RoboDK station: Simulation copy.rdk

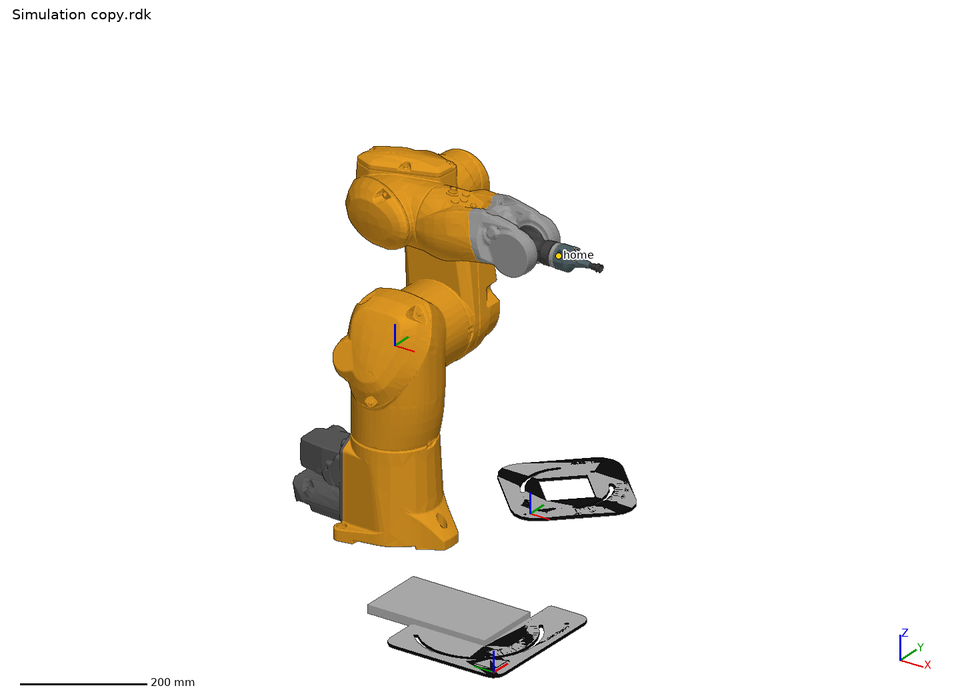
[picture v0: the station drawn from its stored meshes, robots at their saved joint values, targets as dots, program paths as lines]
Station Simulation (saved by RoboDK 5.9.1). Poses are relative to the parent item; angles as X-Y-Z fixed-axis rotations.
  - frame world at (0, 0, 0) mm
    - frame Staubli TX2-40 Base at (0, 0, 0) mm
      - robot Staubli TX2-40: 6 axes, payload 2 kg, reach 515 mm, repeatability 0.02 mm, weight 29 kg
          modified DH rows (alpha deg, a mm, theta deg, d mm): 0, 0, 0, 320; -90, 0, -90, 35; 0, 225, -90, 0; -90, 0, 0, 225; 90, 0, 0, 0; -90, 0, 180, 65
          base shift (0, 0, -320) mm
          joint limits [-180, -180, -180, -270, -180, -270] to [180, 180, 180, 270, 180.5, 270]; home [0, 0, 90, 0, 0, 0]; saved at [0, 0, 90, 0, 0, 0]
        - tool AROB_LWS_VakuumGreifer_14, TCP at (0, 0, 0) mm, size 81.8 x 41.9 x 49.7 mm, geometry from AROB_LWS_VakuumGreifer_14.stp
      - target home (Cartesian target) at (290, 35, 225) mm, rotated rx 0 ry 90 rz 0 deg; joints [0, 0, 90, 0, 0, 0] of Staubli TX2-40
    - frame MagazineFrame at (400, -300, -340) mm, rotated rx 0 ry 0 rz 90 deg
      - object magazinplatte at (100, 100, 0) mm, size 260 x 220 x 5 mm, geometry from AROB_Magazinplatte.stl
      - object jengastuck1 at (72.5, 97.5, 0) mm, rotated rx 0 ry 0 rz 90 deg, size 75 x 25 x 15 mm, geometry from AROB_Jengastuck.stl
      - object jengastuck2 at (97.5, 97.5, 0) mm, rotated rx 0 ry 0 rz 90 deg, size 75 x 25 x 15 mm, geometry from AROB_Jengastuck.stl
      - object jengastuck3 at (122.5, 97.5, 0) mm, rotated rx 0 ry 0 rz 90 deg, size 75 x 25 x 15 mm, geometry from AROB_Jengastuck.stl
      - object jengastuck4 at (147.5, 97.5, 0) mm, rotated rx 0 ry 0 rz 90 deg, size 75 x 25 x 15 mm, geometry from AROB_Jengastuck.stl
      - object jengastuck5 at (172.5, 97.5, 0) mm, rotated rx 0 ry 0 rz 90 deg, size 75 x 25 x 15 mm, geometry from AROB_Jengastuck.stl
      - object jengastuck6 at (72.5, 172.5, 0) mm, rotated rx 0 ry 0 rz 90 deg, size 75 x 25 x 15 mm, geometry from AROB_Jengastuck.stl
      - object jengastuck7 at (97.5, 172.5, 0) mm, rotated rx 0 ry 0 rz 90 deg, size 75 x 25 x 15 mm, geometry from AROB_Jengastuck.stl
      - object jengastuck8 at (122.5, 172.5, 0) mm, rotated rx 0 ry 0 rz 90 deg, size 75 x 25 x 15 mm, geometry from AROB_Jengastuck.stl
      - object jengastuck9 at (147.5, 172.5, 0) mm, rotated rx 0 ry 0 rz 90 deg, size 75 x 25 x 15 mm, geometry from AROB_Jengastuck.stl
      - object jengastuck10 at (172.5, 172.5, 0) mm, rotated rx 0 ry 0 rz 90 deg, size 75 x 25 x 15 mm, geometry from AROB_Jengastuck.stl
      - object jengastuck11 at (72.5, 247.5, 0) mm, rotated rx 0 ry 0 rz 90 deg, size 75 x 25 x 15 mm, geometry from AROB_Jengastuck.stl
      - object jengastuck12 at (97.5, 247.5, 0) mm, rotated rx 0 ry 0 rz 90 deg, size 75 x 25 x 15 mm, geometry from AROB_Jengastuck.stl
      - object jengastuck13 at (122.5, 247.5, 0) mm, rotated rx 0 ry 0 rz 90 deg, size 75 x 25 x 15 mm, geometry from AROB_Jengastuck.stl
      - object jengastuck14 at (147.5, 247.5, 0) mm, rotated rx 0 ry 0 rz 90 deg, size 75 x 25 x 15 mm, geometry from AROB_Jengastuck.stl
      - object jengastuck15 at (172.5, 247.5, 0) mm, rotated rx 0 ry 0 rz 90 deg, size 75 x 25 x 15 mm, geometry from AROB_Jengastuck.stl
    - frame TowerFrame at (120, 200, -340) mm
      - object turmplatte at (0, 100, 0) mm, rotated rx 0 ry 0 rz 45 deg, size 200 x 200 x 5 mm, geometry from AROB_Turmplatte.stl
  - Python program main (listed below)

--- Python program main ---
# main.py

import time
from robodk import robolink

from magazine import Magazine
from tower import Tower
from robot_controller import RobotController
from gripper import Gripper
from jenga_logic import GrabAtPos, ReleaseAtPos

def main():
    # Initialisierung RoboDK API
    rdk = robolink.Robolink()

     # ❗ Kollisionserkennung deaktivieren (nur zum Testen!)
    rdk.setCollisionActive(False)

    # Koordinatenursprünge
    magazine_frame = [330, -100, -300]
    tower_frame = [120, 200, -300]

    # Objekte erzeugen
    magazine = Magazine(magazine_frame)
    tower = Tower(tower_frame)
    robot = RobotController(rdk)
    gripper = Gripper(rdk)

    jenga_pieces = [rdk.Item(f"AROB_Jengastuck{i+1}") for i in range(0,15)]

    for piece in jenga_pieces:
        print(f"Position:{piece.Name()}")



    # Startposition anfahren
    robot.move_to_start()
    robot.move_to_idle()

    # 15 Steine verarbeiten
    for i in range(15):
        source_piece = magazine.get_next_piece()
        source_piece = jenga_pieces[i]
        target_piece = tower.get_next_target(source_piece)

        GrabAtPos(robot, source_piece, gripper)
        ReleaseAtPos(robot, target_piece, gripper)

    # Abschluss
    robot.move_to_start()

if __name__ == "__main__":
    main()
